// TIA Portal project "task3_stateMachine" (V17)

(* hardware
DEVICE "S7-300/ET200M station_1"  S7-300 station
   slot 0: "Rail_0"  Rail  6ES7 390-1***0-0AA0
   slot 2: "PLC_1"  CPU 314C-2 DP  6ES7 314-6CG03-0AB0  V2.6
      slot 0: "MPI interface_1"  X1
      slot 1: "DP interface_1"  X2
      slot 2: "DI 24/DO 16_1"  DI24/DO16
      slot 3: "AI 5/AO 2_1"  AI5/AO2
      slot 4: "Count_1"  Counter
      slot 5: "Positioning_1"  Positioning
*)

// ===== PLC "PLC_1"  CPU 314C-2 DP =====

VAR_GLOBAL   // PLC tag table "Default tag table"
   "start" AT %I0.0 : Bool;
   "FC1" AT %I0.1 : Bool;
   "FC2" AT %I0.2 : Bool;
   "FC3" AT %I0.3 : Bool;
   "FC4" AT %I0.4 : Bool;
   "FC5" AT %I0.5 : Bool;
   "Normal_motor" AT %Q0.0 : Bool;
   "Low_speed_motor" AT %Q0.1 : Bool;
   "Reverse_motor" AT %Q0.2 : Bool;
   "Piston" AT %Q0.3 : Bool;
   "G1" AT %I0.6 : Bool;
   "G2" AT %I0.7 : Bool;
   "flag1" AT %M4.0 : Bool;
   "flag2" AT %M4.1 : Bool;
   "flag3" AT %M4.2 : Bool;
   "flag4" AT %M4.3 : Bool;
END_VAR

ORGANIZATION_BLOCK "Main"   // OB1, LAD
TITLE = "Main Program Sweep (Cycle)"
{ S7_Optimized_Access := 'FALSE' }
VERSION : 0.1
   VAR_TEMP
      OB1_EV_CLASS : Byte;   // Bits 0-3 = 1 (Coming event), Bits 4-7 = 1 (Event class 1)
      OB1_SCAN_1 : Byte;   // 1 (Cold restart scan 1 of OB 1), 3 (Scan 2-n of OB 1)
      OB1_PRIORITY : Byte;   // Priority of OB Execution
      OB1_OB_NUMBR : Byte;   // 1 (Organization block 1, OB1)
      OB1_RESERVED_1 : Byte;   // Reserved for system
      OB1_RESERVED_2 : Byte;   // Reserved for system
      OB1_PREV_CYCLE : Int;   // Cycle time of previous OB1 scan (milliseconds)
      OB1_MIN_CYCLE : Int;   // Minimum cycle time of OB1 (milliseconds)
      OB1_MAX_CYCLE : Int;   // Maximum cycle time of OB1 (milliseconds)
      OB1_DATE_TIME : Date_And_Time;   // Date and time OB1 started
   END_VAR
BEGIN

REGION Network 1: starts conveyor normally
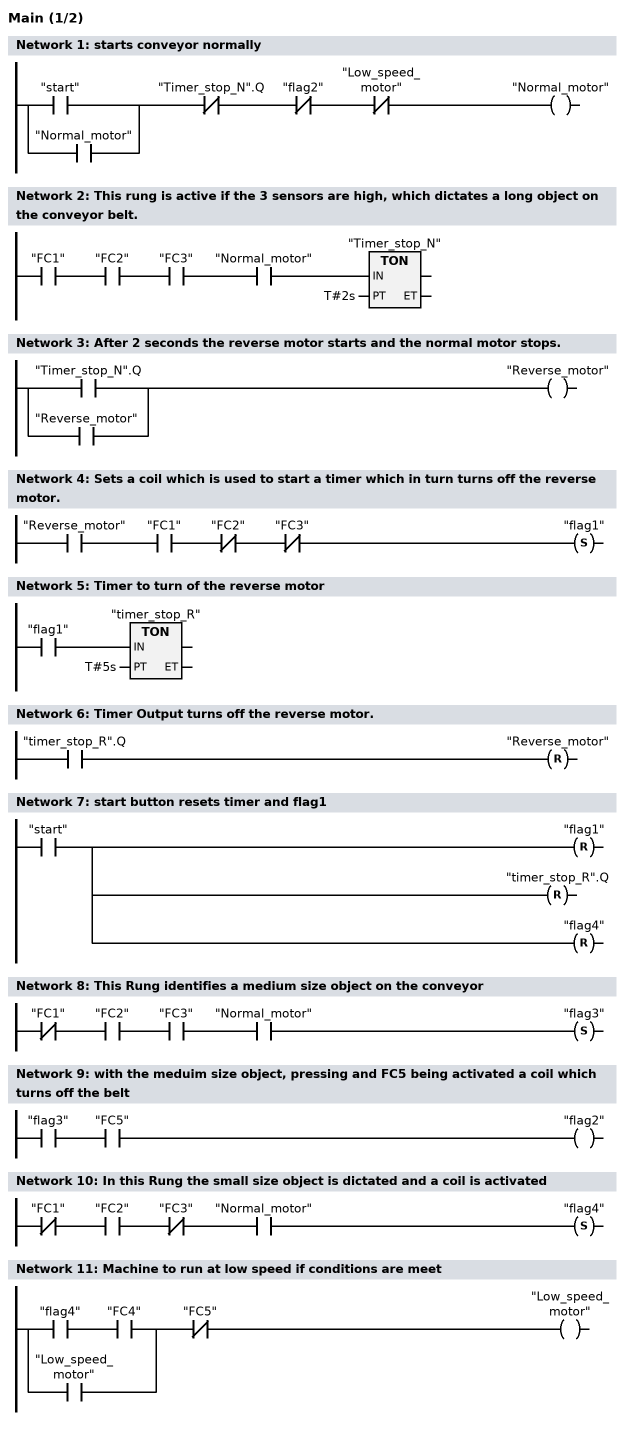
   RUNG wire#powerrail
      Contact( "start" )
      wire#w1
      I_Contact( "Timer_stop_N".Q )
      I_Contact( "flag2" )
      I_Contact( "Low_speed_motor" )
      Coil( "Normal_motor" )
   END_RUNG
   RUNG wire#powerrail
      Contact( "Normal_motor" )
   END_RUNG wire#w1
   // the same network as SCL:
   "Normal_motor" := ("start" OR "Normal_motor") AND NOT "Timer_stop_N".Q AND NOT "flag2" AND NOT "Low_speed_motor";
END_REGION

REGION Network 2: This rung is active if the 3 sensors are high, which dictates a long object on the conveyor belt.
   "Timer_stop_N".TON(IN := "FC1" AND "FC2" AND "FC3" AND "Normal_motor", PT := T#2s);
END_REGION

REGION Network 3: After 2 seconds the reverse motor starts and the normal motor stops.
   RUNG wire#powerrail
      Contact( "Timer_stop_N".Q )
      wire#w1
      Coil( "Reverse_motor" )
   END_RUNG
   RUNG wire#powerrail
      Contact( "Reverse_motor" )
   END_RUNG wire#w1
   // the same network as SCL:
   "Reverse_motor" := "Timer_stop_N".Q OR "Reverse_motor";
END_REGION

REGION Network 4: Sets a coil which is used to start a timer which in turn turns off the reverse motor.
   RUNG wire#powerrail
      Contact( "Reverse_motor" )
      Contact( "FC1" )
      I_Contact( "FC2" )
      I_Contact( "FC3" )
      S_Coil( "flag1" )
   END_RUNG
   // the same network as SCL:
   IF "Reverse_motor" AND "FC1" AND NOT "FC2" AND NOT "FC3" THEN "flag1" := TRUE; END_IF;
END_REGION

REGION Network 5: Timer to turn of the reverse motor
   "timer_stop_R".TON(IN := "flag1", PT := T#5s);
END_REGION

REGION Network 6: Timer Output turns off the reverse motor.
   RUNG wire#powerrail
      Contact( "timer_stop_R".Q )
      R_Coil( "Reverse_motor" )
   END_RUNG
   // the same network as SCL:
   IF "timer_stop_R".Q THEN "Reverse_motor" := FALSE; END_IF;
END_REGION

REGION Network 7: start button resets timer and flag1
   RUNG wire#powerrail
      Contact( "start" )
      wire#w1
      R_Coil( "flag1" )
   END_RUNG
   RUNG wire#w1
      R_Coil( "timer_stop_R".Q )
   END_RUNG
   RUNG wire#w1
      R_Coil( "flag4" )
   END_RUNG
   // the same network as SCL:
   IF "start" THEN
       "flag1" := FALSE;
       "timer_stop_R".Q := FALSE;
       "flag4" := FALSE;
   END_IF;
END_REGION

REGION Network 8: This Rung identifies a medium size object on the conveyor
   RUNG wire#powerrail
      I_Contact( "FC1" )
      Contact( "FC2" )
      Contact( "FC3" )
      Contact( "Normal_motor" )
      S_Coil( "flag3" )
   END_RUNG
   // the same network as SCL:
   IF NOT "FC1" AND "FC2" AND "FC3" AND "Normal_motor" THEN "flag3" := TRUE; END_IF;
END_REGION

REGION Network 9: with the meduim size object, pressing and FC5 being activated a coil which turns off the belt
   RUNG wire#powerrail
      Contact( "flag3" )
      Contact( "FC5" )
      Coil( "flag2" )
   END_RUNG
   // the same network as SCL:
   "flag2" := "flag3" AND "FC5";
END_REGION

REGION Network 10: In this Rung the small size object is dictated and a coil is activated
   RUNG wire#powerrail
      I_Contact( "FC1" )
      Contact( "FC2" )
      I_Contact( "FC3" )
      Contact( "Normal_motor" )
      S_Coil( "flag4" )
   END_RUNG
   // the same network as SCL:
   IF NOT "FC1" AND "FC2" AND NOT "FC3" AND "Normal_motor" THEN "flag4" := TRUE; END_IF;
END_REGION

REGION Network 11: Machine to run at low speed if conditions are meet
   RUNG wire#powerrail
      Contact( "flag4" )
      Contact( "FC4" )
      wire#w1
      I_Contact( "FC5" )
      Coil( "Low_speed_motor" )
   END_RUNG
   RUNG wire#powerrail
      Contact( "Low_speed_motor" )
   END_RUNG wire#w1
   // the same network as SCL:
   "Low_speed_motor" := (("flag4" AND "FC4") OR "Low_speed_motor") AND NOT "FC5";
END_REGION

REGION Network 12
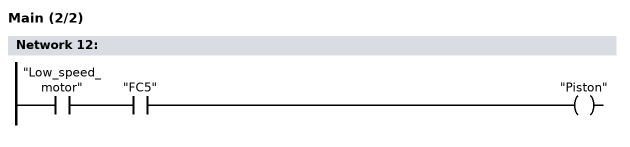
   RUNG wire#powerrail
      Contact( "Low_speed_motor" )
      Contact( "FC5" )
      Coil( "Piston" )
   END_RUNG
   // the same network as SCL:
   "Piston" := "Low_speed_motor" AND "FC5";
END_REGION
END_ORGANIZATION_BLOCK